TYPE "Positioning_EPOS_Machine_Manager"
VERSION : 0.1
// Block: Positioning_EPOS_Machine_Manager
   STRUCT
      EnableStopDoorOpeningReq : Bool;
      EnableStopInPhase : Bool;
      EnableStopProgrammed : Bool;
      Control_ON : Bool;
      Minus : Bool;
      Plus : Bool;
      MoveToPos : Bool;
      Pos : LReal;
      Vel : LReal;
      Acc : LReal;
      Dec : LReal;
   END_STRUCT;

END_TYPE
